// Funzione che ritorna TRUE se almeno un WORKFLOW è in errore
FUNCTION TFIsWorkflowError : BOOL 
VAR_INPUT
	WorkFlow : POINTER TO ARRAY[0..MAXWORKFLOW] OF WorkFlow;
END_VAR
VAR
	i: UINT;
END_VAR

FOR i:=0 TO MAXWORKFLOW DO
	IF WorkFlow^[i].State = StateWF_ERROR THEN
		TFIsWorkflowError := TRUE;
		RETURN;
	END_IF
END_FOR

END_FUNCTION

(* stored: Version 1.1.0.1, ProductVersion 3.1.4024.11
   POU TFIsWorkflowError: Id {becf03c7-6334-406a-970a-9de1e737d573}, SpecialFunc None *)
